// TIA Portal project "G120" (V20)

(* hardware
DEVICE "SINAMICS G_1"  Sinamics.Device
   slot 0: "	_0"  Rail  SinamicsG120RackPN
   slot 0: "Drive"  G120 CU240E-2 PN-F  6SL3244-0BB13-1FA0  4.5
      slot 1: "PROFINET interface"  MDD-SinamicsG120-P
   slot 3: "PM240 IP20"  PM240 IP20  6SL3224-0BE13-7UA0  -
DEVICE "S7-1500/ET200MP station_1"  S7-1500 station
   slot 0: "Rail_0"  Rack  6ES7 590-1***0-0AA0
   slot 1: "Brain"  CPU 1511C-1 PN  6ES7 511-1CK00-0AB0  V2.5
      slot 3: "CPU display_1"  6ES7591-1AA00-0AA0
      slot 32768: "PROFINET interface_1"  X1
         slot 32769: "Port_1"  X1 P1
         slot 32770: "Port_2"  X1 P2
*)

// ===== PLC "Brain"  CPU 1511C-1 PN =====

VAR_GLOBAL   // PLC tag table "Default tag table"
   "Tag_1" AT %M0.0 : Bool;
END_VAR

VAR_GLOBAL   // PLC tag table "Motor Data"
   "Motor Setpoint Speed" AT %QW258 : Int;
   "Motor Potentiometer" AT %MW40 : Int;
   "Normalized Speed" AT %MD42 : Real;
   "Clearance_0" AT %Q256.2 : Bool;
   "Clearance_1" AT %Q257.1 : Bool;
   "Clearance_2" AT %Q257.2 : Bool;
   "Clearance_3" AT %Q257.3 : Bool;
   "Clearance_4" AT %Q257.4 : Bool;
   "Clearance_5" AT %Q257.5 : Bool;
   "Clearance_6" AT %Q257.6 : Bool;
   "Clearance_7" AT %Q257.7 : Bool;
   "Motor ON" AT %Q256.0 : Bool;
   "Motor ON Push Button" AT %I2.0 : Bool;
   "Reverse Motor Switch" AT %I2.1 : Bool;
   "Reverse Motor" AT %Q256.3 : Bool;
END_VAR

FUNCTION "Motor" : Void   // FC1, LAD
{ S7_Optimized_Access := 'TRUE' }
VERSION : 0.1
BEGIN

REGION Network 1
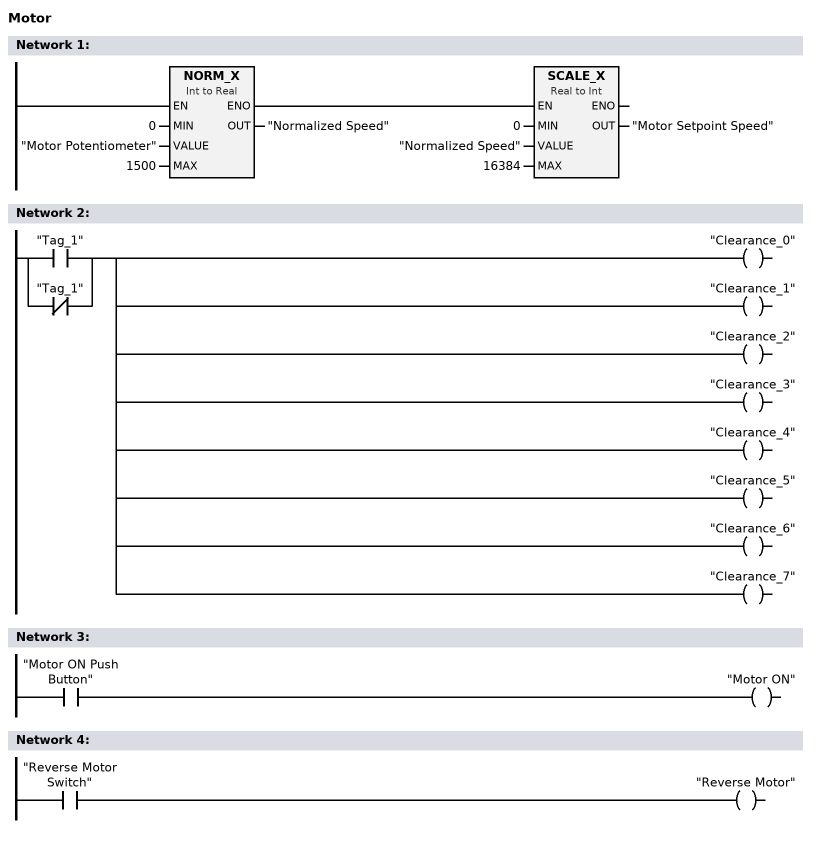
   RUNG wire#powerrail
      { S7_Templates := "[SrcType := Int, DestType := Real]" } Normalize(min := 0, value := "Motor Potentiometer", max := 1500, out => "Normalized Speed")
      { S7_Templates := "[SrcType := Real, DestType := Int]" } Scale(min := 0, value := "Normalized Speed", max := 16384, out => "Motor Setpoint Speed")
   END_RUNG
   // the same network as SCL:
   "Normalized Speed" := NORM_X(MIN := 0, VALUE := "Motor Potentiometer", MAX := 1500);
   "Motor Setpoint Speed" := SCALE_X(MIN := 0, VALUE := "Normalized Speed", MAX := 16384);
END_REGION

REGION Network 2
   RUNG wire#powerrail
      Contact( "Tag_1" )
      wire#w1
      Coil( "Clearance_0" )
   END_RUNG
   RUNG wire#powerrail
      I_Contact( "Tag_1" )
   END_RUNG wire#w1
   RUNG wire#w1
      Coil( "Clearance_1" )
   END_RUNG
   RUNG wire#w1
      Coil( "Clearance_2" )
   END_RUNG
   RUNG wire#w1
      Coil( "Clearance_3" )
   END_RUNG
   RUNG wire#w1
      Coil( "Clearance_4" )
   END_RUNG
   RUNG wire#w1
      Coil( "Clearance_5" )
   END_RUNG
   RUNG wire#w1
      Coil( "Clearance_6" )
   END_RUNG
   RUNG wire#w1
      Coil( "Clearance_7" )
   END_RUNG
   // the same network as SCL:
   "Clearance_0" := "Tag_1" OR NOT "Tag_1";
   "Clearance_1" := "Clearance_0";
   "Clearance_2" := "Clearance_0";
   "Clearance_3" := "Clearance_0";
   "Clearance_4" := "Clearance_0";
   "Clearance_5" := "Clearance_0";
   "Clearance_6" := "Clearance_0";
   "Clearance_7" := "Clearance_0";
END_REGION

REGION Network 3
   RUNG wire#powerrail
      Contact( "Motor ON Push Button" )
      Coil( "Motor ON" )
   END_RUNG
   // the same network as SCL:
   "Motor ON" := "Motor ON Push Button";
END_REGION

REGION Network 4
   RUNG wire#powerrail
      Contact( "Reverse Motor Switch" )
      Coil( "Reverse Motor" )
   END_RUNG
   // the same network as SCL:
   "Reverse Motor" := "Reverse Motor Switch";
END_REGION
END_FUNCTION

ORGANIZATION_BLOCK "Main"   // OB1, LAD, ProgramCycle
TITLE = "Main Program Sweep (Cycle)"
{ S7_Optimized_Access := 'TRUE' }
VERSION : 0.1
   VAR_INPUT
      Initial_Call : Bool;   // Initial call of this OB
      Remanence : Bool;   // =True, if remanent data are available
   END_VAR
BEGIN

REGION Network 1
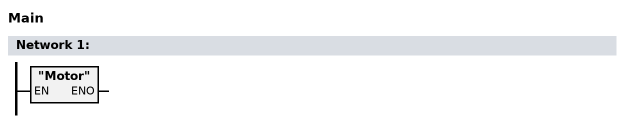
   RUNG wire#powerrail
      "Motor"()
   END_RUNG
   // the same network as SCL:
   "Motor"();
END_REGION
END_ORGANIZATION_BLOCK